ABB RobotStudio station: mesa-paletizadora2026.rspag

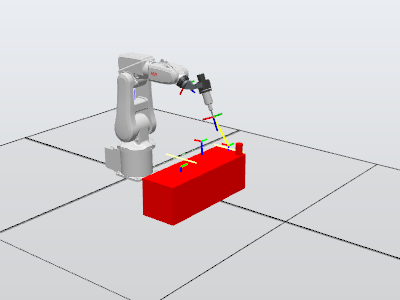
--- station ---
Station mesa-paletizadora2026 (saved by RobotStudio 25.3.11371.0)
Controller IRB120_3_58
  mechanical unit ROB_1: IRB120_3_58__01, 6 joints, base frame (0, 0, 0) mm
Layout (positions relative to the parent item):
  - IRB120_3_58__01 [mechanism, from %ABB.RobotStudio.Models.IRB120%\IRB120_3_58_G_01.rslib] at (0, 0, 0) mm; joint values [0, 0, 0, 0, 0.5236, 0] (rad or m)
  - MyTool [mechanism, from Training Objects\myTool.rslib] at (364.35, 0, 594) mm, rotated rx 180 ry 60 rz 180 deg
  - MESA [smart component]
      signals: DI MOVER_MESA, DI COLOR
      connections:
        MESA.MOVER_MESA -> LinearMover2.Execute
        MESA.COLOR -> Highlighter_3.Active
    - mesa [part] at (400, -380, 0) mm, size 204.9 x 607.3 x 204.9 mm
    - LinearMover2 [smart component, from Components\LinearMover2.rslib]
        properties: Object=mesa; Direction=[0 -0.001 0]; Distance=0.08; Duration=1; Reference=Global; ReferenceObject=(none)
    - Highlighter_3 [smart component, from Components\Highlighter.rslib]
        properties: Object=mesa; Color=[50 50 100]; Opacity=255
  - fotocelulas [smart component]
      signals: DO cajaEnOrigen, DO CajaTercera
      connections:
        LineSensor.SensorOut -> fotocelulas.cajaEnOrigen
        LineSensor_2.SensorOut -> fotocelulas.CajaTercera
    - LineSensor [smart component, from Components\LineSensor.rslib]
        properties: Start=[0.4 0.2 0.215]; End=[0.6 0.2 0.215]; Length=0.2; Radius=0; Tag=(none); SenseMultiple=false; SensedPart=baliza; SensedPoint=[0.5567705078125 0.2 0.215]
      - _sensorPart_ [part], size 200 x 0 x 0 mm
    - LineSensor_2 [smart component, from Components\LineSensor.rslib]
        properties: Start=[0.4 -0.2 0.275]; End=[0.6 -0.2 0.275]; Length=0.2; Radius=0; Tag=(none); SenseMultiple=false; SensedPart=(none); SensedPoint=[0 0 0]
      - _sensorPart_ [part], size 200 x 0 x 0 mm
  - CONTROL_CAJA [smart component]
      signals: DI Sacar_caja, DI habilitar, DI ventosa, DO colision
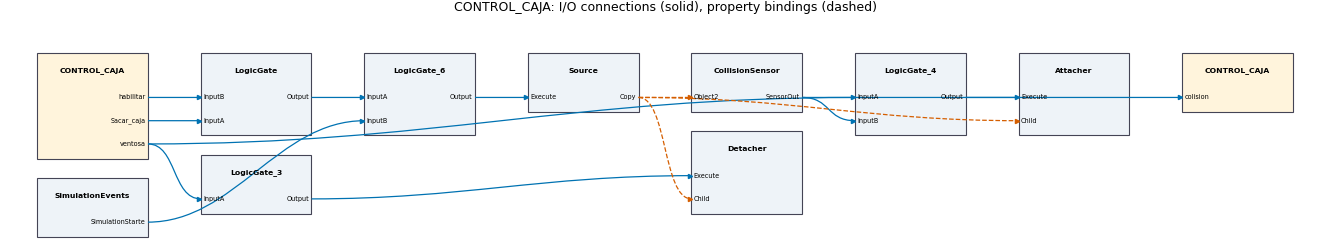
      connections:
        CONTROL_CAJA.habilitar -> LogicGate.InputB
        CONTROL_CAJA.Sacar_caja -> LogicGate.InputA
        LogicGate_3.Output -> Detacher.Execute
        CONTROL_CAJA.ventosa -> LogicGate_3.InputA
        CollisionSensor.SensorOut -> CONTROL_CAJA.colision
        CONTROL_CAJA.ventosa -> LogicGate_4.InputA
        CollisionSensor.SensorOut -> LogicGate_4.InputB
        LogicGate_4.Output -> Attacher.Execute
        LogicGate.Output -> LogicGate_6.InputA
        SimulationEvents.SimulationStarted -> LogicGate_6.InputB
        LogicGate_6.Output -> Source.Execute
        Source.Copy => Attacher.Child
        Source.Copy => Detacher.Child
        Source.Copy => CollisionSensor.Object2
    - Source [smart component, from Components\Source.rslib]
        properties: Source=caja; Copy=(none); Parent=(none); Position=[0.5 0.2 0.2]; Orientation=[0 0 0]; Transient=true; PhysicsBehavior=3
    - caja [part], size 50.8 x 40.5 x 30.9 mm
    - LogicGate [smart component, from Components\LogicGate.rslib]
        properties: Operator=AND; Delay=0
    - Attacher [smart component, from Components\Attacher.rslib]
        properties: Parent=MyTool; Flange=0; Child=(none); Mount=false; Offset=[0 0 0]; Orientation=[0 0 0]
    - Detacher [smart component, from Components\Detacher.rslib]
        properties: Child=(none); KeepPosition=true
    - LogicGate_3 [smart component, from Components\LogicGate.rslib]
        properties: Operator=NOT; Delay=0
    - CollisionSensor [smart component, from Components\CollisionSensor.rslib]
        properties: Object1=MyTool; Object2=(none); NearMiss=0.002; Part1=(none); Part2=(none); CollisionType=0
      - _sensorPart_ [part]
    - LogicGate_4 [smart component, from Components\LogicGate.rslib]
        properties: Operator=AND; Delay=0
    - LogicGate_5 [smart component, from Components\LogicGate.rslib]
        properties: Operator=OR; Delay=0
    - SimulationEvents [smart component, from Components\SimulationEvents.rslib]
    - SimulationEvents_2 [smart component, from Components\SimulationEvents.rslib]
    - LogicGate_6 [smart component, from Components\LogicGate.rslib]
        properties: Operator=OR; Delay=0
  - baliza [smart component]
      signals: DI encender
      connections:
        baliza.encender -> Highlighter.Active
    - baliza [part] at (-1.08, -75.93, 1.22) mm, rotated rx 0 ry 0 rz -0.22 deg, size 40 x 39.9 x 60 mm
    - Highlighter [smart component, from Components\Highlighter.rslib]
        properties: Object=baliza; Color=[0 255 0]; Opacity=255
Attachment: MyTool is attached to IRB120_3_58__01 / Link6
Station signals: DI MOVER_MESA, DI SACAR_CAJA, DI MARCHA, DO CajaEnOrigen, DO habilitar, DO ventosa, DO colision, DO CajaTercera
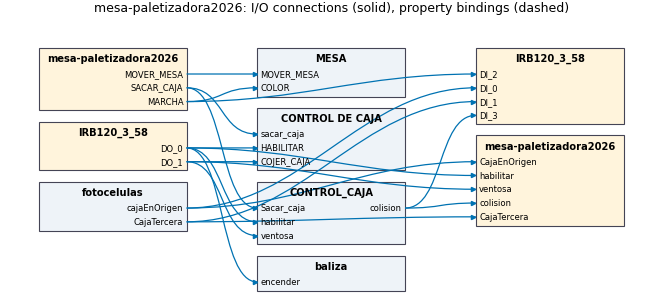
Station logic (signal -> signal, property => property):
  mesa-paletizadora2026.MOVER_MESA -> MESA.MOVER_MESA
  mesa-paletizadora2026.SACAR_CAJA -> CONTROL DE CAJA.sacar_caja
  IRB120_3_58.DO_0 -> CONTROL DE CAJA.HABILITAR
  IRB120_3_58.DO_1 -> CONTROL DE CAJA.COJER_CAJA
  mesa-paletizadora2026.MARCHA -> IRB120_3_58.DI_2
  fotocelulas.cajaEnOrigen -> mesa-paletizadora2026.CajaEnOrigen
  fotocelulas.cajaEnOrigen -> IRB120_3_58.DI_0
  IRB120_3_58.DO_0 -> mesa-paletizadora2026.habilitar
  mesa-paletizadora2026.SACAR_CAJA -> CONTROL_CAJA.Sacar_caja
  IRB120_3_58.DO_0 -> CONTROL_CAJA.habilitar
  IRB120_3_58.DO_1 -> mesa-paletizadora2026.ventosa
  IRB120_3_58.DO_1 -> CONTROL_CAJA.ventosa
  CONTROL_CAJA.colision -> mesa-paletizadora2026.colision
  fotocelulas.CajaTercera -> IRB120_3_58.DI_1
  fotocelulas.CajaTercera -> mesa-paletizadora2026.CajaTercera
  CONTROL_CAJA.colision -> IRB120_3_58.DI_3
  IRB120_3_58.DO_0 -> baliza.encender
  mesa-paletizadora2026.MARCHA -> MESA.COLOR
Targets, tools, work objects and paths stored in the station and not in the controller backup, written as RAPID:
! task T_ROB1
MODULE Module1
  CONST robtarget Target_10:=[[547.330665099,0,451.64730631],[0.190808996,0,0.981627183,0],[0,0,0,0],[9E+09,9E+09,9E+09,9E+09,9E+09,9E+09]];
  CONST robtarget Target_20:=[[471.959035864,0,303.311229798],[0.024300739,0,0.999704693,0],[0,0,0,0],[9E+09,9E+09,9E+09,9E+09,9E+09,9E+09]];
ENDMODULE


--- Controller Data/IRB120_3_58/RAPID/TASK1/PROGMOD/CalibData.mod ---
MODULE CalibData
    PERS tooldata MyTool:=[TRUE,[[31.7926,0,229.639],[0.945519,0,0.325568,0]],[1,[0,0,1],[1,0,0,0],0,0,0]];
    TASK PERS wobjdata Workobject_1:=[FALSE,TRUE,"",[[0,0,0],[1,0,0,0]],[[0,0,0],[1,0,0,0]]];
ENDMODULE

--- Controller Data/IRB120_3_58/RAPID/TASK1/PROGMOD/Module1.mod ---
MODULE Module1
    CONST robtarget inicio:=[[547.330665099,0,451.64730631],[0.190808996,0,0.981627183,0],[0,0,0,0],[9E+09,9E+09,9E+09,9E+09,9E+09,9E+09]];

    CONST robtarget centro_caja:=[[500,200,230],[0,0,1,0],[0,-1,0,0],[9E+09,9E+09,9E+09,9E+09,9E+09,9E+09]];
    CONST robtarget caja_desplazada:=[[500,-200,230],[0,0,1,0],[0,-1,0,0],[9E+09,9E+09,9E+09,9E+09,9E+09,9E+09]];
    VAR num ALTURA:=0;

    VAR num cajas:=0;    !altura de la caja 30mm
!ENTRADAS
    !DI_0 sensor caja en origen
    !DI_1 sensor caja tercera colocada
    !DI_2 pulsador de marcha
       !DI_3 Colision
!SALIDAS
    !D0_0 habilitar sacar caja
    !D0_1 ventosa
    PROC main()
        MoveL inicio,v800,z100,MyTool\WObj:=Workobject_1;
        Set DO_0;! habilitar sacar caja
        WaitDI DI_2,1;! espera a poner el selector a 1


        WaitTime 1;       !tienes 3 segundos para añadir una caja
        ReSet DO_0;       !deshabilitar sacar caja
         MoveLDo centro_caja,v400,z0,MyTool\WObj:=Workobject_1,DO_1,1; !vete a la caja y activa la ventosa
         WaitTime 1;

         IF di_3=1  THEN!si cogemos una caja

            cajas:=cajas+1;
             IF cajas=7 THEN  !inicializo los contadores y vuelvo a empezar
                       ALTURA:=0;
                       cajas:=0;
                   ENDIF
                 IF cajas<4 THEN
                        Path_10;
                        ALTURA:=ALTURA+40;
                  ENDIF
                  IF cajas=4 ALTURA:=0;
                  IF  cajas>=4 AND cajas<7  THEN

                    Path_20;
                    ALTURA:=ALTURA+40;
                  ENDIF

             WaitTime 1;
            Reset DO_1; !Suelta la caja
        ELSE !si no tiene caja vuelve a inicio y resetea valores
                reset DO_1;
              cajas:=0;
              ALTURA:=0;

         ENDIF



    ENDPROC

    PROC Path_10()

        MoveL inicio,v800,z100,MyTool\WObj:=Workobject_1;
        MoveL Offs(caja_desplazada,0,0,ALTURA),v400,z0,MyTool\WObj:=Workobject_1;
    ENDPROC

     PROC Path_20()

        MoveL inicio,v800,z100,MyTool\WObj:=Workobject_1;
        MoveL Offs(caja_desplazada,0,40,ALTURA),v400,z0,MyTool\WObj:=Workobject_1;
    ENDPROC

ENDMODULE

--- Controller Data/IRB120_3_58/SYSPAR/EIO.cfg ---
EIO:CFG_1.0:6:1::
#
INDUSTRIAL_NETWORK:

      -Name "DeviceNet" -Label "DeviceNet Master/Slave Network" -Address "2"
#
DEVICENET_DEVICE:

      -Name "d652" -VendorName "ABB Robotics" -ProductName "24 VDC I/O Device"\
      -Label "DSQC 652 24 VDC I/O Device" -Address 10 -ProductCode 26\
      -DeviceType 7 -ConnectionType "COS" -OutputSize 2 -InputSize 2
#
DEVICENET_INTERNAL_DEVICE:

      -Name "DN_Internal_Device" -VendorName "ABB Robotics"\
      -ProductName "DeviceNet Internal Slave Device"
#
EIO_SIGNAL:

      -Name "DI_0" -SignalType "DI" -Device "d652" -DeviceMap "0" -Access "All"

      -Name "DI_1" -SignalType "DI" -Device "d652" -DeviceMap "1" -Access "All"

      -Name "DI_2" -SignalType "DI" -Device "d652" -DeviceMap "2" -Access "All"

      -Name "DI_3" -SignalType "DI" -Device "d652" -DeviceMap "3" -Access "All"

      -Name "DI_4" -SignalType "DI" -Device "d652" -DeviceMap "4" -Access "All"

      -Name "DI_5" -SignalType "DI" -Device "d652" -DeviceMap "5" -Access "All"

      -Name "DO_0" -SignalType "DO" -Device "d652" -DeviceMap "0" -Access "All"

      -Name "DO_1" -SignalType "DO" -Device "d652" -DeviceMap "1" -Access "All"

      -Name "DO_2" -SignalType "DO" -Device "d652" -DeviceMap "2" -Access "All"

      -Name "DO_3" -SignalType "DO" -Device "d652" -DeviceMap "3" -Access "All"

      -Name "DO_4" -SignalType "DO" -Device "d652" -DeviceMap "4" -Access "All"

      -Name "DO_5" -SignalType "DO" -Device "d652" -DeviceMap "5" -Access "All"
